(*
Manages the lifecycle and transitions of states within an entity.  
Supports queuing state change requests, triggering state transitions, and broadcasting state change events.  
Adds a `_stateChangeEvent` Signal to the owning `I_Entity` during initialization, enabling external components to listen for state changes.
*)
FUNCTION_BLOCK FINAL StateManager IMPLEMENTS I_Execute, I_StateManager, I_Debug

VAR
	_comp				: Component(THIS^);

	_exe				: Execute(THIS^);
	_sm					: _StateMachine;
	_buffer				: _StateBuffer;
	
	_stateChangeEvent	: Signal;
	
	_iPretender			: I_State;
	_iCurrent			: I_State;
	_iPrevious 			: I_State;
	
	
END_VAR

(*
Retrieves the currently active state managed by the state manager.
*)
PROPERTY Current : I_State
GET
Current := _iCurrent;
END_GET
END_PROPERTY

// DO NOT CALL MANUALLY
{attribute 'hide'}
METHOD Execute
VAR_INPUT
	nPhase: INT := 0;
END_VAR
VAR
	_iNewState		: I_StateInternal;
	_iOldState		: I_StateInternal;
END_VAR
IF IsOk(_buffer.Pop(iState => _iNewState)) THEN
	_iPretender := _iNewState._AsIState;
	IF IsOk(_sm.Change(_iNewState, iOldState => _iOldState)) THEN
		_stateChangeEvent.Emit(_iNewState._AsIState.Tag);
		
		_iCurrent		:= _iNewState._AsIState;
		IF _iOldState <> 0 THEN
			_iPrevious		:= _iOldState._AsIState;
		END_IF
		
	END_IF
	
	_iPretender		:= 0;
END_IF
END_METHOD

(*
Returns the entity that owns this state.
*)
PROPERTY Owner : I_Entity
GET
Owner := _comp.Entity;
END_GET
END_PROPERTY

(*
Retrieves the state that is queued to become active next, but has not yet transitioned.
*)
PROPERTY Pretender : I_State
GET
Pretender := _iPretender;
END_GET
END_PROPERTY

(*
Retrieves the last active state prior to the current one.
*)
PROPERTY Previous : I_State
GET
Previous := _iPrevious;
END_GET
END_PROPERTY

(*
Allows initializing an external interface variable with an interface pointer to this instance within declaration block.
Example:
iSMgr: I_StateManager;
smgr: StateManager := (Proxy := iSMgr);
Result: iSMgr <> 0 
*)
PROPERTY Proxy : REFERENCE TO I_StateManager
SET
Proxy := THIS^;
END_SET
END_PROPERTY

(*
Queues a request to transition to a specified state.  
Returns:
- `Ok` - If the state change request is successfully queued.
- `Err.Itf0` - If the provided state interface is invalid.
- `Err.NoMatch` - If the state does not belong to the same entity.
- `Err.IncArg` - If the state is already in the queue.
*)
METHOD Request : Result
VAR_INPUT
	iState			: I_State;
END_VAR
VAR
	iStateInternal	: I_StateInternal;
END_VAR
IF iState = 0 THEN
	Request := Err.Itf0;
	RETURN;
END_IF

IF iState.Owner <> _comp.Entity THEN
	Request := Err.NoMatch;
	RETURN;
END_IF

Request := _buffer.Push(iState._AsIStateInternal);
END_METHOD

END_FUNCTION_BLOCK

(* stored: Version 1.1.0.1
   POU StateManager: Id {9af5d38b-2c9a-4ad2-afd9-0321b459f566}, SpecialFunc None
   Folder _: Id {b9f442f7-4971-4185-be3d-d4d6b1569cc6}
   Folder Request: Id {81375855-59e4-4ae6-b079-7f9366b0efcb}
   Folder State: Id {3323aa43-3a83-405c-9127-b99e6e5b1777}
   Property Current: Id {56420e57-ba0a-40d3-a86e-12a2b1e27f6c}
   Get Get: Id {6dfc2ef8-549f-4ef6-9ab0-969a1aced6b1}
   Method Execute: Id {f267a716-e453-4e52-a04a-1da93f557d85}
   Property Owner: Id {f4018121-2b1d-444e-9a31-6e2d9cde72f4}
   Get Get: Id {f50d6afe-6131-4b10-8754-fbb6797dbc8d}
   Property Pretender: Id {03d469e9-e5de-4b22-9ad6-7121be122863}
   Get Get: Id {cd77ba45-868a-497f-86a5-d426aa5face8}
   Property Previous: Id {506a1524-211d-46a2-a335-40f8e25eab3e}
   Get Get: Id {34c2f99f-f5d0-4f3c-a7e7-87b5355c4a6f}
   Property Proxy: Id {c84b4b1b-1dde-471a-9a35-21636f83c5d3}
   Set Set: Id {f44529b5-5fa8-4582-ba32-00ad5d0d8de7}
   Method Request: Id {12dc1eaf-0190-483f-ada2-8afa12a43cbf} *)
